PROGRAM P_Demo_FB_GetLicenseDongles
VAR
    fbFB_GetLicenseDongles : FB_GetLicenseDongles; // FB_GetLicenseDongles 实例
    bExec                  : BOOL := FALSE;
    bBusy_                 : BOOL;
    bErrFlag               : BOOL;
    nErrCode               : UDINT;
END_VAR

// =============================================================================
// 场景：多 dongle 列出。
// 价值：多 dongle 环境管理。
// 验证：触发后观察 bDone / bErr，错误号 nErrId 反映 ADS Return Codes。
// 验证步骤：
//   1. 右键 PLC 项目下 POUs 文件夹 → Add → Existing Item → 选本 .TcPOU 文件
//   2. 引用 Tc2_Utilities（References → Add library）
//   3. 编译 → 登录 → 运行；按上方『验证』行的指示在线写值观察
// =============================================================================

fbFB_GetLicenseDongles(
    bExecute := bExec, tTimeout := DEFAULT_ADS_TIMEOUT,
    bBusy => bBusy_, bError => bErrFlag, nErrorId => nErrCode
);

END_PROGRAM

(* stored: Version 1.1.0.1, ProductVersion 3.1.4024.5
   POU P_Demo_FB_GetLicenseDongles: Id {74e802ce-a2c2-5479-a660-357f93b2c6d9}, SpecialFunc None *)
